{attribute 'GeneratedUsingTerminal: EP2816-0004-0016'}
{attribute addProperty BoxType "EP2816-0004-0016"}
{attribute addProperty Description "EP2816-0004 16 Ch. Dig. Output 24V, 0,5A, M16"}
{attribute addProperty Physics "YY"}
{attribute addProperty Id "DO_Outputs_Channel_1AT %Q*DO_Outputs_Channel_28AC1A9E8DO_Outputs_Channel_2AT %Q*DO_Outputs_Channel_28AC1A9E8WcStateAT %I*WcState_0B2B16F91InfoDataAT %I*InfoData_32EB74EA10"}
{attribute addProperty CRC "2284994867"}
{attribute addProperty Size "27"}
TYPE EP2816_88324133 EXTENDS EtcSlaveBoxBase_77A0E4A7 :
STRUCT
	{attribute addProperty Name "DO_Outputs_Channel_1"}
	DO_Outputs_Channel_1 : DO_Outputs_Channel_28AC1A9E;
	{attribute addProperty Name "DO_Outputs_Channel_2"}
	DO_Outputs_Channel_2 : DO_Outputs_Channel_28AC1A9E;
	{attribute addProperty Name "WcState"}
	WcState : WcState_0B2B16F9;
	{attribute addProperty Name "InfoData"}
	InfoData : InfoData_32EB74EA;
END_STRUCT
END_TYPE

(* stored: Version 1.2.0.0, ProductVersion 3.1.4024.11
   DUT EP2816_88324133: Id {673a865e-1638-4f62-b981-1cf5eae1d8fb} *)
